{attribute 'GeneratedUsingTerminal: AT2041-0250-0023'}
{attribute addProperty BoxType "AT2041-0250-0023"}
{attribute addProperty Id "A_0099_AT2040_5250_0018_AT2040_5250AT2040_01D6DEDF80"}
{attribute addProperty CRC "3277424192"}
{attribute addProperty Size "80"}
TYPE A_0045_AT2041_0250_0023_C3598640 EXTENDS AT2041_86175B41 :
STRUCT
	{attribute addProperty Name "A_0099_AT2040_5250_0018_AT2040_5250"}
	{attribute addProperty PreviousPort "A_0045(AT2041-0250-0023) : B"}
	A_0099_AT2040_5250_0018_AT2040_5250 : AT2040_01D6DEDF;
END_STRUCT
END_TYPE

(* stored: Version 1.2.0.0, ProductVersion 3.1.4024.9
   DUT A_0045_AT2041_0250_0023_C3598640: Id {71ac0ac5-118d-4b5c-aec7-3c1dc781dedd} *)
